// TIA Portal V17 export
// export: Created 2025-06-26T06:33:55.1370113Z, ExportSetting WithDefaults, DisplayName Totally Integrated Automation Portal, DisplayVersion V17 Update 8, DisplayName TIA Portal Openness, DisplayVersion V17 Update 8, DisplayName TIA Portal Version Control Interface, DisplayVersion V17, DisplayName STEP 7 Professional, DisplayVersion V17 Update 8, DisplayName STEP 7 Safety, DisplayVersion V17 Update 6, DisplayName WinCC Advanced, DisplayVersion V17 Update 8
FUNCTION "fcCustomerMapping" : Void   // FC1, FBD
TITLE = Map IO tags to DBs
{ S7_Optimized_Access := 'TRUE' }
VERSION : 0.1
// stored: AutoNumber true, IsIECCheckEnabled false, SetENOAutomatically false, UDAEnableTagReadback false
BEGIN

REGION Network 1 (SCL): Comments
   // If using S7 communication with the customer, use DB_ToHB & DB_FromHB
   // If not, still move everything into these DBs, but then use this block for copying to/from I/O memory
   // Also, the DBs can contain a superset of those things actually sent or received (S7 communication has higher bandwidth)
   // Could also be in its own OB, just like Modbus, so it can "feed into" DB_ToHB and DB_FromHB transparently
END_REGION

REGION Network 2 (SCL): Signals in from customer ("ToHb")
   // Commands
   //"DB_ToHB".StartRequest := "VB3-M8301 Start";

   // Customer-specific signals
   //"DB_ToHB".Setpoint := "ScaleIn"(nIn := "QI117_828B1");
END_REGION

REGION Network 3 (SCL): Signals out to Customer ("FromHB")
   // Status bits
   //"VB3-M8301 NA-Status"   := "DB_FromHB".EmergencyStopStatus;
END_REGION
END_FUNCTION
